ABB RobotStudio station: TPL01.rsstnx

Station Project2 (saved by RobotStudio 25.5.11605.0)
Controller IRB140_6_81
  mechanical unit ROB_1: IRB140_6_81_C_03, 6 joints, base frame (0, 0, 0) mm
Layout (positions relative to the parent item):
  - IRB140_6_81_C_03 [mechanism, from %ABB.RobotStudio.Models.IRB140%\IRB140_6_81_C_G_03.rslib] at (0, 0, 0) mm; joint values [-0.1496, -0.0274, 0.4762, 2.8072, 0.4714, -2.4487] (rad or m)
  - Mesa [part], size 365 x 405 x 340 mm
  - Perno [part] at (730, 340, 177) mm, rotated rx 90 ry 0 rz -90 deg, size 20 x 100 x 20 mm
  - Pinza [mechanism] at (463, -60, 547) mm, rotated rx 90 ry 67.5 rz 90 deg
      TCP Pinza at (0, 0, 137) mm, rotated rx 0 ry 0 rz -22.5 deg
      links: Dummy
Attachment: Pinza is attached to IRB140_6_81_C_03 / Link6
Attachment: REF_Mesa is attached to Mesa
Attachment: REF_perno is attached to Perno
EventTableEntry 2314: ActivationMode=2, Cyclic=false, Group=, Trigger=DO_Pinza 2315, Actions=[EventTableActionAttach 2316], Comment=
EventTableTriggerIO 2315: Operator=0, IOValue=[1], IRC5Controller=? -1, SignalSource=IRB140_6_81 1261
EventTableActionAttach 2316: MountObject=false, FlangeIndext=0, FindNearest=false, AttachmentParent=Pinza 2308, AttachmentChild=Perno 2304, Offset=[X=1, Y=0, Z=0, W=0, X=0, Y=1, Z=0, W=0, X=0, Y=0, Z=1, W=0, X=0, Y=0, Z=0, W=1]
EventTableEntry 2317: ActivationMode=2, Cyclic=false, Group=, Trigger=DO_Pinza 2318, Actions=[EventTableActionDetach 2319], Comment=
EventTableTriggerIO 2318: Operator=0, IOValue=[0], IRC5Controller=? -1, SignalSource=IRB140_6_81 1261
EventTableActionDetach 2319: AttachmentParent=Pinza 2308, AttachmentChild=Perno 2304
Collision set CollisionSet_1: Perno against Mesa, near miss 0.005 m
EventTableTriggerIO 2517: Operator=0, IOValue=[1], IRC5Controller=? -1, SignalSource=IRB140_6_81 1261
EventTableTriggerIO 2518: Operator=0, IOValue=[0], IRC5Controller=? -1, SignalSource=IRB140_6_81 1261
Targets, tools, work objects and paths stored in the station, written as RAPID:
! task T_ROB1
MODULE CalibData
  PERS tooldata Pinza:=[TRUE,[[0,0,137],[0.98078528,0,0,-0.195090322]],[0.5,[0,0,100],[1,0,0,0],0,0,0]];
  TASK PERS wobjdata REF_Mesa:=[FALSE,TRUE,"",[[665,-400,260],[0,0,1,0]],[[0,0,0],[1,0,0,0]]];
  TASK PERS wobjdata REF_perno:=[FALSE,TRUE,"",[[359.999760413,-259.999933044,129.999820452],[0.500000242,0.500000092,0.499999436,0.500000231]],[[0,0,0],[1,0,0,0]]];
ENDMODULE

! task T_ROB1
MODULE Module1
  CONST robtarget TOMAR_PIEZA:=[[0,0,10],[0.5,0.5,-0.5,0.5],[0,0,0,0],[9E+09,9E+09,9E+09,9E+09,9E+09,9E+09]];
  CONST robtarget INSERTAR_PIEZA:=[[65,340,3],[1,0,0,0],[-1,1,-2,0],[9E+09,9E+09,9E+09,9E+09,9E+09,9E+09]];
  PERS tooldata TCP_perno:=[TRUE,[[0,0,227],[0.980785,0,0,-0.19509]],[0.5,[0,0,100],[1,0,0,0],0,0,0]];
  CONST robtarget home_10:=[[624.937,0,611],[1,0,0,0],[0,0,0,0],[9E+09,9E+09,9E+09,9E+09,9E+09,9E+09]];
  PROC test_path()
    SetDO DO_Pinza,0;
    MoveJ Offs(TOMAR_PIEZA,0,offset1,0),v1000,fine,Pinza\WObj:=REF_Perno;
    MoveL TOMAR_PIEZA,v1000,fine,Pinza\WObj:=REF_Perno;
    SetDO DO_Pinza,1;
    MoveL Offs(TOMAR_PIEZA,0,offset2,0),v1000,fine,Pinza\WObj:=REF_Perno;
    MoveJ Offs(INSERTAR_PIEZA,0,0, -offset3),v1000,fine,TCP_perno\WObj:=REF_Mesa;
    MoveL INSERTAR_PIEZA,v1000,fine,TCP_perno\WObj:=REF_Mesa;
    SetDO DO_Pinza,0;
    MoveL Offs(INSERTAR_PIEZA,0,0, -offset3),v1000,fine,TCP_perno\WObj:=REF_Mesa;
  ENDPROC
  PROC main()
    test_path;
  ENDPROC
ENDMODULE

